{attribute 'GeneratedUsingTerminal: EK1100-0000-0018'}
{attribute addProperty BoxType "EK1100-0000-0018"}
{attribute addProperty Id "Beckhoff_EL67xxEK1122Beckhoff_EL67xxEK1122_4856750E2A_0001_EL6720_0000_0016EL6720_210A1A8D16A_0002_EL6720_0000_0017EL6720_210A1A8D16A_0003_EL6720_0000_0018EL6720_210A1A8D16A_0004_EL6720_0000_0020EL6720_210A1A8D16A_0005_EL6731_0000_0000EL6731_210A1A8D16A_0006_EL6731_0001_0000EL6731_210A1A8D16A_0007_EL6731_0000_0016EL6731_210A1A8D16A_0008_EL6731_0000_0017EL6731_210A1A8D16A_0009_EL6731_0000_0018EL6731_210A1A8D16A_0010_EL6731_0000_0019EL6731_210A1A8D16A_0011_EL6731_0000_0020EL6731_210A1A8D16A_0012_EL6731_0000_0021EL6731_210A1A8D16A_0013_EL6731_0000_0022EL6731_210A1A8D16A_0014_EL6731_0000_0023EL6731_210A1A8D16A_0015_EL6731_0000_0025EL6731_210A1A8D16A_0016_EL6731_0100_0017EL6731_210A1A8D16A_0017_EL6731_0100_0018EL6731_210A1A8D16A_0018_EL6731_0100_0019EL6731_210A1A8D16A_0019_EL6731_0100_0020EL6731_210A1A8D16A_0020_EL6731_0100_0021EL6731_210A1A8D16A_0021_EL6731_0100_0022EL6731_210A1A8D16A_0022_EL6731_0100_0023EL6731_210A1A8D16A_0023_EL6731_0100_0025EL6731_210A1A8D16A_0024_EL6731_0010_0000EL6731_210A1A8D16A_0025_EL6731_0010_0016EL6731_210A1A8D16A_0026_EL6731_0010_0017EL6731_210A1A8D16A_0027_EL6731_0010_0018EL6731_210A1A8D16A_0028_EL6731_0010_0019EL6731_210A1A8D16A_0029_EL6731_0010_0021EL6731_210A1A8D16A_0030_EL6731_1003_0016EL6731_210A1A8D16A_0031_EL6740_0010_0000EL6740_BB2AF53012A_0032_EL6740_0010_0001EL6740_BB2AF53012A_0033_EL6740_0010_0002EL6740_BB2AF53012A_0034_EL6751_0000_0000EL6751_210A1A8D16A_0035_EL6751_0001_0000EL6751_210A1A8D16A_0036_EL6751_0000_0016EL6751_210A1A8D16A_0037_EL6751_0000_0017EL6751_210A1A8D16A_0038_EL6751_0000_0018EL6751_210A1A8D16A_0039_EL6751_0000_0019EL6751_210A1A8D16A_0040_EL6751_0000_0021EL6751_210A1A8D16A_0041_EL6751_0000_0022EL6751_210A1A8D16A_0042_EL6751_0005_0022EL6751_210A1A8D16A_0043_EL6751_0010_0000EL6751_210A1A8D16A_0044_EL6751_0010_0017EL6751_210A1A8D16A_0045_EL6751_0010_0018EL6751_210A1A8D16A_0046_EL6751_0010_0019EL6751_210A1A8D16A_0047_EL6751_0010_0021EL6751_210A1A8D16A_0048_EL6752_0000_0000EL6752_210A1A8D16A_0049_EL6752_0000_0016EL6752_210A1A8D16A_0050_EL6752_0000_0017EL6752_210A1A8D16A_0051_EL6752_0000_0018EL6752_210A1A8D16A_0052_EL6752_0000_0019EL6752_210A1A8D16A_0053_EL6752_0000_0020EL6752_210A1A8D16A_0054_EL6752_0010_0000EL6752_210A1A8D16A_0055_EL6752_0010_0016EL6752_210A1A8D16A_0056_EL6752_0010_0017EL6752_210A1A8D16A_0057_EL6752_0010_0018EL6752_210A1A8D16A_0058_EL6752_0010_0020EL6752_210A1A8D16A_0059_EL6784_0000_0016EL6784_9D61BA3F16A_0060_EL6784_0000_0017EL6784_9D61BA3F16A_0061_EL6784_0000_0018EL6784_9D61BA3F16"}
{attribute addProperty CRC "2634234538"}
{attribute addProperty Size "966"}
TYPE Beckhoff_EL67xx_9D033AAA EXTENDS EK1100_1FC0878B :
STRUCT
	{attribute addProperty Name "Beckhoff_EL67xxEK1122"}
	{attribute addProperty PreviousPort "Beckhoff EL67xx : B"}
	Beckhoff_EL67xxEK1122 : Beckhoff_EL67xxEK1122_4856750E;
	{attribute addProperty Name "A_0001_EL6720_0000_0016"}
	{attribute addProperty PreviousPort "Beckhoff EL67xxEK1122 : C"}
	A_0001_EL6720_0000_0016 : EL6720_210A1A8D;
	{attribute addProperty Name "A_0002_EL6720_0000_0017"}
	{attribute addProperty PreviousPort "A_0001(EL6720-0000-0016) : B"}
	A_0002_EL6720_0000_0017 : EL6720_210A1A8D;
	{attribute addProperty Name "A_0003_EL6720_0000_0018"}
	{attribute addProperty PreviousPort "A_0002(EL6720-0000-0017) : B"}
	A_0003_EL6720_0000_0018 : EL6720_210A1A8D;
	{attribute addProperty Name "A_0004_EL6720_0000_0020"}
	{attribute addProperty PreviousPort "A_0003(EL6720-0000-0018) : B"}
	A_0004_EL6720_0000_0020 : EL6720_210A1A8D;
	{attribute addProperty Name "A_0005_EL6731_0000_0000"}
	{attribute addProperty PreviousPort "A_0004(EL6720-0000-0020) : B"}
	A_0005_EL6731_0000_0000 : EL6731_210A1A8D;
	{attribute addProperty Name "A_0006_EL6731_0001_0000"}
	{attribute addProperty PreviousPort "A_0005(EL6731-0000-0000) : B"}
	A_0006_EL6731_0001_0000 : EL6731_210A1A8D;
	{attribute addProperty Name "A_0007_EL6731_0000_0016"}
	{attribute addProperty PreviousPort "A_0006(EL6731-0001-0000) : B"}
	A_0007_EL6731_0000_0016 : EL6731_210A1A8D;
	{attribute addProperty Name "A_0008_EL6731_0000_0017"}
	{attribute addProperty PreviousPort "A_0007(EL6731-0000-0016) : B"}
	A_0008_EL6731_0000_0017 : EL6731_210A1A8D;
	{attribute addProperty Name "A_0009_EL6731_0000_0018"}
	{attribute addProperty PreviousPort "A_0008(EL6731-0000-0017) : B"}
	A_0009_EL6731_0000_0018 : EL6731_210A1A8D;
	{attribute addProperty Name "A_0010_EL6731_0000_0019"}
	{attribute addProperty PreviousPort "A_0009(EL6731-0000-0018) : B"}
	A_0010_EL6731_0000_0019 : EL6731_210A1A8D;
	{attribute addProperty Name "A_0011_EL6731_0000_0020"}
	{attribute addProperty PreviousPort "A_0010(EL6731-0000-0019) : B"}
	A_0011_EL6731_0000_0020 : EL6731_210A1A8D;
	{attribute addProperty Name "A_0012_EL6731_0000_0021"}
	{attribute addProperty PreviousPort "A_0011(EL6731-0000-0020) : B"}
	A_0012_EL6731_0000_0021 : EL6731_210A1A8D;
	{attribute addProperty Name "A_0013_EL6731_0000_0022"}
	{attribute addProperty PreviousPort "A_0012(EL6731-0000-0021) : B"}
	A_0013_EL6731_0000_0022 : EL6731_210A1A8D;
	{attribute addProperty Name "A_0014_EL6731_0000_0023"}
	{attribute addProperty PreviousPort "A_0013(EL6731-0000-0022) : B"}
	A_0014_EL6731_0000_0023 : EL6731_210A1A8D;
	{attribute addProperty Name "A_0015_EL6731_0000_0025"}
	{attribute addProperty PreviousPort "A_0014(EL6731-0000-0023) : B"}
	A_0015_EL6731_0000_0025 : EL6731_210A1A8D;
	{attribute addProperty Name "A_0016_EL6731_0100_0017"}
	{attribute addProperty PreviousPort "A_0015(EL6731-0000-0025) : B"}
	A_0016_EL6731_0100_0017 : EL6731_210A1A8D;
	{attribute addProperty Name "A_0017_EL6731_0100_0018"}
	{attribute addProperty PreviousPort "A_0016(EL6731-0100-0017) : B"}
	A_0017_EL6731_0100_0018 : EL6731_210A1A8D;
	{attribute addProperty Name "A_0018_EL6731_0100_0019"}
	{attribute addProperty PreviousPort "A_0017(EL6731-0100-0018) : B"}
	A_0018_EL6731_0100_0019 : EL6731_210A1A8D;
	{attribute addProperty Name "A_0019_EL6731_0100_0020"}
	{attribute addProperty PreviousPort "A_0018(EL6731-0100-0019) : B"}
	A_0019_EL6731_0100_0020 : EL6731_210A1A8D;
	{attribute addProperty Name "A_0020_EL6731_0100_0021"}
	{attribute addProperty PreviousPort "A_0019(EL6731-0100-0020) : B"}
	A_0020_EL6731_0100_0021 : EL6731_210A1A8D;
	{attribute addProperty Name "A_0021_EL6731_0100_0022"}
	{attribute addProperty PreviousPort "A_0020(EL6731-0100-0021) : B"}
	A_0021_EL6731_0100_0022 : EL6731_210A1A8D;
	{attribute addProperty Name "A_0022_EL6731_0100_0023"}
	{attribute addProperty PreviousPort "A_0021(EL6731-0100-0022) : B"}
	A_0022_EL6731_0100_0023 : EL6731_210A1A8D;
	{attribute addProperty Name "A_0023_EL6731_0100_0025"}
	{attribute addProperty PreviousPort "A_0022(EL6731-0100-0023) : B"}
	A_0023_EL6731_0100_0025 : EL6731_210A1A8D;
	{attribute addProperty Name "A_0024_EL6731_0010_0000"}
	{attribute addProperty PreviousPort "A_0023(EL6731-0100-0025) : B"}
	A_0024_EL6731_0010_0000 : EL6731_210A1A8D;
	{attribute addProperty Name "A_0025_EL6731_0010_0016"}
	{attribute addProperty PreviousPort "A_0024(EL6731-0010-0000) : B"}
	A_0025_EL6731_0010_0016 : EL6731_210A1A8D;
	{attribute addProperty Name "A_0026_EL6731_0010_0017"}
	{attribute addProperty PreviousPort "A_0025(EL6731-0010-0016) : B"}
	A_0026_EL6731_0010_0017 : EL6731_210A1A8D;
	{attribute addProperty Name "A_0027_EL6731_0010_0018"}
	{attribute addProperty PreviousPort "A_0026(EL6731-0010-0017) : B"}
	A_0027_EL6731_0010_0018 : EL6731_210A1A8D;
	{attribute addProperty Name "A_0028_EL6731_0010_0019"}
	{attribute addProperty PreviousPort "A_0027(EL6731-0010-0018) : B"}
	A_0028_EL6731_0010_0019 : EL6731_210A1A8D;
	{attribute addProperty Name "A_0029_EL6731_0010_0021"}
	{attribute addProperty PreviousPort "A_0028(EL6731-0010-0019) : B"}
	A_0029_EL6731_0010_0021 : EL6731_210A1A8D;
	{attribute addProperty Name "A_0030_EL6731_1003_0016"}
	{attribute addProperty PreviousPort "A_0029(EL6731-0010-0021) : B"}
	A_0030_EL6731_1003_0016 : EL6731_210A1A8D;
	{attribute addProperty Name "A_0031_EL6740_0010_0000"}
	{attribute addProperty PreviousPort "A_0030(EL6731-1003-0016) : B"}
	A_0031_EL6740_0010_0000 : EL6740_BB2AF530;
	{attribute addProperty Name "A_0032_EL6740_0010_0001"}
	{attribute addProperty PreviousPort "A_0031(EL6740-0010-0000) : B"}
	A_0032_EL6740_0010_0001 : EL6740_BB2AF530;
	{attribute addProperty Name "A_0033_EL6740_0010_0002"}
	{attribute addProperty PreviousPort "A_0032(EL6740-0010-0001) : B"}
	A_0033_EL6740_0010_0002 : EL6740_BB2AF530;
	{attribute addProperty Name "A_0034_EL6751_0000_0000"}
	{attribute addProperty PreviousPort "A_0033(EL6740-0010-0002) : B"}
	A_0034_EL6751_0000_0000 : EL6751_210A1A8D;
	{attribute addProperty Name "A_0035_EL6751_0001_0000"}
	{attribute addProperty PreviousPort "A_0034(EL6751-0000-0000) : B"}
	A_0035_EL6751_0001_0000 : EL6751_210A1A8D;
	{attribute addProperty Name "A_0036_EL6751_0000_0016"}
	{attribute addProperty PreviousPort "A_0035(EL6751-0001-0000) : B"}
	A_0036_EL6751_0000_0016 : EL6751_210A1A8D;
	{attribute addProperty Name "A_0037_EL6751_0000_0017"}
	{attribute addProperty PreviousPort "A_0036(EL6751-0000-0016) : B"}
	A_0037_EL6751_0000_0017 : EL6751_210A1A8D;
	{attribute addProperty Name "A_0038_EL6751_0000_0018"}
	{attribute addProperty PreviousPort "A_0037(EL6751-0000-0017) : B"}
	A_0038_EL6751_0000_0018 : EL6751_210A1A8D;
	{attribute addProperty Name "A_0039_EL6751_0000_0019"}
	{attribute addProperty PreviousPort "A_0038(EL6751-0000-0018) : B"}
	A_0039_EL6751_0000_0019 : EL6751_210A1A8D;
	{attribute addProperty Name "A_0040_EL6751_0000_0021"}
	{attribute addProperty PreviousPort "A_0039(EL6751-0000-0019) : B"}
	A_0040_EL6751_0000_0021 : EL6751_210A1A8D;
	{attribute addProperty Name "A_0041_EL6751_0000_0022"}
	{attribute addProperty PreviousPort "A_0040(EL6751-0000-0021) : B"}
	A_0041_EL6751_0000_0022 : EL6751_210A1A8D;
	{attribute addProperty Name "A_0042_EL6751_0005_0022"}
	{attribute addProperty PreviousPort "A_0041(EL6751-0000-0022) : B"}
	A_0042_EL6751_0005_0022 : EL6751_210A1A8D;
	{attribute addProperty Name "A_0043_EL6751_0010_0000"}
	{attribute addProperty PreviousPort "A_0042(EL6751-0005-0022) : B"}
	A_0043_EL6751_0010_0000 : EL6751_210A1A8D;
	{attribute addProperty Name "A_0044_EL6751_0010_0017"}
	{attribute addProperty PreviousPort "A_0043(EL6751-0010-0000) : B"}
	A_0044_EL6751_0010_0017 : EL6751_210A1A8D;
	{attribute addProperty Name "A_0045_EL6751_0010_0018"}
	{attribute addProperty PreviousPort "A_0044(EL6751-0010-0017) : B"}
	A_0045_EL6751_0010_0018 : EL6751_210A1A8D;
	{attribute addProperty Name "A_0046_EL6751_0010_0019"}
	{attribute addProperty PreviousPort "A_0045(EL6751-0010-0018) : B"}
	A_0046_EL6751_0010_0019 : EL6751_210A1A8D;
	{attribute addProperty Name "A_0047_EL6751_0010_0021"}
	{attribute addProperty PreviousPort "A_0046(EL6751-0010-0019) : B"}
	A_0047_EL6751_0010_0021 : EL6751_210A1A8D;
	{attribute addProperty Name "A_0048_EL6752_0000_0000"}
	{attribute addProperty PreviousPort "A_0047(EL6751-0010-0021) : B"}
	A_0048_EL6752_0000_0000 : EL6752_210A1A8D;
	{attribute addProperty Name "A_0049_EL6752_0000_0016"}
	{attribute addProperty PreviousPort "A_0048(EL6752-0000-0000) : B"}
	A_0049_EL6752_0000_0016 : EL6752_210A1A8D;
	{attribute addProperty Name "A_0050_EL6752_0000_0017"}
	{attribute addProperty PreviousPort "A_0049(EL6752-0000-0016) : B"}
	A_0050_EL6752_0000_0017 : EL6752_210A1A8D;
	{attribute addProperty Name "A_0051_EL6752_0000_0018"}
	{attribute addProperty PreviousPort "A_0050(EL6752-0000-0017) : B"}
	A_0051_EL6752_0000_0018 : EL6752_210A1A8D;
	{attribute addProperty Name "A_0052_EL6752_0000_0019"}
	{attribute addProperty PreviousPort "A_0051(EL6752-0000-0018) : B"}
	A_0052_EL6752_0000_0019 : EL6752_210A1A8D;
	{attribute addProperty Name "A_0053_EL6752_0000_0020"}
	{attribute addProperty PreviousPort "A_0052(EL6752-0000-0019) : B"}
	A_0053_EL6752_0000_0020 : EL6752_210A1A8D;
	{attribute addProperty Name "A_0054_EL6752_0010_0000"}
	{attribute addProperty PreviousPort "A_0053(EL6752-0000-0020) : B"}
	A_0054_EL6752_0010_0000 : EL6752_210A1A8D;
	{attribute addProperty Name "A_0055_EL6752_0010_0016"}
	{attribute addProperty PreviousPort "A_0054(EL6752-0010-0000) : B"}
	A_0055_EL6752_0010_0016 : EL6752_210A1A8D;
	{attribute addProperty Name "A_0056_EL6752_0010_0017"}
	{attribute addProperty PreviousPort "A_0055(EL6752-0010-0016) : B"}
	A_0056_EL6752_0010_0017 : EL6752_210A1A8D;
	{attribute addProperty Name "A_0057_EL6752_0010_0018"}
	{attribute addProperty PreviousPort "A_0056(EL6752-0010-0017) : B"}
	A_0057_EL6752_0010_0018 : EL6752_210A1A8D;
	{attribute addProperty Name "A_0058_EL6752_0010_0020"}
	{attribute addProperty PreviousPort "A_0057(EL6752-0010-0018) : B"}
	A_0058_EL6752_0010_0020 : EL6752_210A1A8D;
	{attribute addProperty Name "A_0059_EL6784_0000_0016"}
	{attribute addProperty PreviousPort "A_0058(EL6752-0010-0020) : B"}
	A_0059_EL6784_0000_0016 : EL6784_9D61BA3F;
	{attribute addProperty Name "A_0060_EL6784_0000_0017"}
	{attribute addProperty PreviousPort "A_0059(EL6784-0000-0016) : B"}
	A_0060_EL6784_0000_0017 : EL6784_9D61BA3F;
	{attribute addProperty Name "A_0061_EL6784_0000_0018"}
	{attribute addProperty PreviousPort "A_0060(EL6784-0000-0017) : B"}
	A_0061_EL6784_0000_0018 : EL6784_9D61BA3F;
END_STRUCT
END_TYPE

(* stored: Version 1.2.0.0, ProductVersion 3.1.4024.9
   DUT Beckhoff_EL67xx_9D033AAA: Id {02618704-8822-4a2e-9ebd-a05b91fe4034} *)
